// LS Electric XG5000 project: 8_29_문제2
// PLC LSPLC
// module base 0 slot 0: 입출력 모듈:XBC-DR14E (DC 24V 입력 8점, 릴레이 출력 6점)

PROGRAM NewProgram (task: 스캔 프로그램)

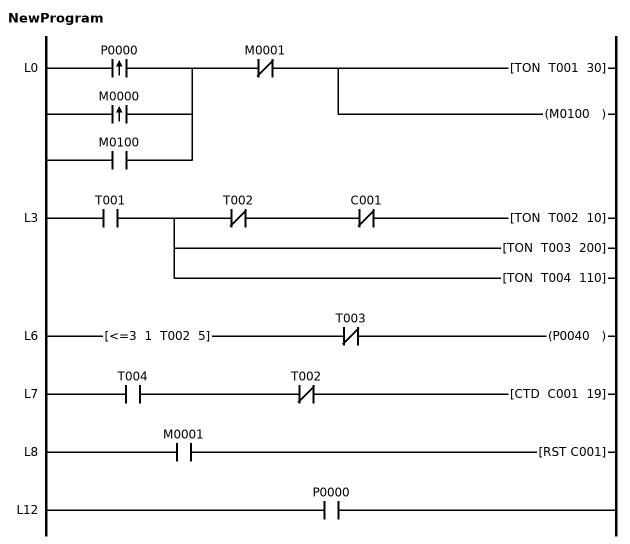
; L0
LOADP     P0000
ORP       M0000
OR        M0100
AND NOT   M0001
TON       T001 30
OUT       M0100
; L3
LOAD      T001
MPUSH
AND NOT   T002
AND NOT   C001
TON       T002 10
MPOP
TON       T003 200
TON       T004 110
; L6
LOAD<=3   1 T002 5
AND NOT   T003
OUT       P0040
; L7
LOAD      T004
AND NOT   T002
CTD       C001 19
; L8
LOAD      M0001
RST       C001
; L12
LOAD      P0000